FUNCTION StringBeginsWith : BOOL
VAR_INPUT
	text : T_MaxString;
	startsWithString : T_MaxString;
END_VAR
VAR
	textLength : DINT;
	length : DINT;
END_VAR

textLength := LEN(text);
length := LEN(startsWithString);

IF (textLength < length) THEN
	RETURN;
END_IF

StringBeginsWith := MEMCMP(pBuf1 := ADR(text), pBuf2 := ADR(startsWithString), n := TO_UDINT(length)) = 0;

END_FUNCTION

(* stored: Version 1.1.0.1
   POU StringBeginsWith: Id {ad6f003b-91a3-0195-1c5a-34153d758fe5}, SpecialFunc None *)
